Universal Robots PolyScope program: whisk_matcha.urp

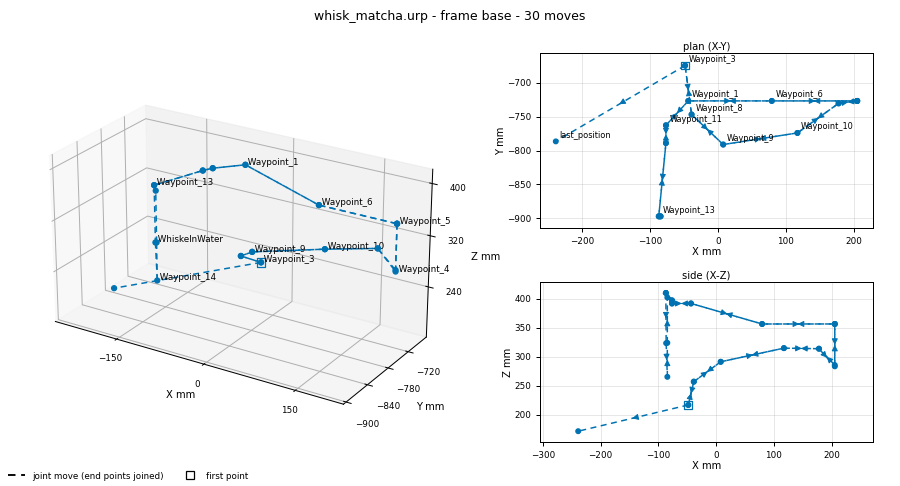
[picture p0: tool path of whisk_matcha.urp in frame base, 30 of 31 moves have a stored position in this frame; points joined in program order, loops and branches not executed]
Program whisk_matcha (installation=default directory=/programs/Matcha createdIn=5.12.6.1102099 lastSavedIn=5.12.6.1102099 robotSerialNumber=20215500597)
Calibrated DH parameters: a=[0.000193, -0.066673, -0.391568, -0.000012, 0.00005, 0]; d=[0.162643, -472.05677, 465.132521, 7.058239, 0.099746, 0.099582]; alpha=[1.571116, 0.00089, 0.003862, 1.569269, -1.569248, 0]; deltaTheta=[0, -1.413394, 7.628392, 0.068187, 0, -0.000001]
Robot Program (runOnlyOnce=true)
  URCap Gripper Activate (Robotiq_Grippers, Robotiq Inc.) dataModel(ResetAndActivateKey=false)
  URCap Gripper (Robotiq_Grippers, Robotiq Inc.) dataModel(position=14.117647058823529, force=0.0, speed=0.0, positionInDouble=14.117647058823529, forceInDouble=0.0, speedInDouble=0.0, slaveIds=[9], blocking=true)
  MoveJ speed 60 deg/s, acceleration 80 deg/s^2 (useActiveTCP=true) feature=Base
    Waypoint Waypoint (Variable): variable=matchaSpoonHome
    Waypoint Waypoint_3: TCP in base x=-48.218 y=-674.691 z=216.535 mm, rx=-1.0956 ry=1.5728 rz=-1.3161 rad; joints [49.709, -52.645, 74.816, -42.693, -23.853, -158.617] deg; TCP offset x=0 y=0 z=191.5 mm, rx=0 ry=0 rz=0 rad
    Waypoint Waypoint_8: TCP in base x=-38.666 y=-746.861 z=256.872 mm, rx=-0.5003 ry=1.6808 rz=-0.7695 rad; joints [54.631, -40.792, 48.492, -25.129, -23.202, -120.249] deg
    Waypoint Waypoint_9: TCP in base x=7.915 y=-791.123 z=291.294 mm, rx=0.1007 ry=1.6659 rz=-0.1248 rad; joints [60.017, -27.831, 19.708, -5.925, -22.495, -78.296] deg
    Waypoint Waypoint_10: TCP in base x=117.298 y=-774.028 z=314.897 mm, rx=0.8846 ry=1.446 rz=0.7971 rad; joints [67.52, -9.771, -20.402, 20.84, -21.505, -19.839] deg
    Waypoint Waypoint_2: TCP in base x=177.976 y=-730.441 z=313.913 mm, rx=1.2449 ry=1.2572 rz=1.2232 rad; joints [71.064, -1.234, -39.351, 33.486, -21.04, 7.782] deg
    Waypoint Waypoint_4: TCP in base x=205.418 y=-726.808 z=283.401 mm, rx=1.2448 ry=1.2573 rz=1.2232 rad; joints [73.018, 4.06, -46.322, 34.472, -19.107, 8.52] deg
  URCap Gripper (Robotiq_Grippers, Robotiq Inc.) dataModel(position=100.0, force=100.0, speed=64.0, positionInDouble=100.0, forceInDouble=100.0, speedInDouble=64.0, slaveIds=[9], blocking=true)
  MoveJ speed 60 deg/s, acceleration 80 deg/s^2 (useActiveTCP=true) feature=Base
    Waypoint Waypoint_5: TCP in base x=205.369 y=-726.831 z=356.753 mm, rx=1.2449 ry=1.2572 rz=1.2232 rad; joints [73.015, -6.018, -35.971, 34.181, -19.107, 8.543] deg
    Waypoint Waypoint_6: TCP in base x=79.554 y=-726.833 z=356.715 mm, rx=1.2449 ry=1.2572 rz=1.2232 rad; joints [63.962, -12.783, -20.178, 27.557, -28.074, 5.907] deg
    Waypoint Waypoint_1: TCP in base x=-43.538 y=-726.812 z=392.259 mm, rx=1.3602 ry=1.0584 rz=1.0356 rad; joints [53.28, -11.873, -28.744, 34.319, -24.003, 6.898] deg
    Waypoint Waypoint_11: TCP in base x=-76.429 y=-762.764 z=392.203 mm, rx=1.4056 ry=0.9656 rz=0.9484 rad; joints [51.982, -14.289, -22.965, 29.233, -18.545, 8.768] deg
    Waypoint Waypoint_18: TCP in base x=-76.468 y=-788.93 z=397.596 mm, rx=1.4283 ry=0.9152 rz=0.9007 rad; joints [52.819, -15.443, -21.159, 26.101, -14.083, 11.353] deg
    Waypoint Waypoint_13: TCP in base x=-87.04 y=-896.924 z=410.452 mm, rx=1.4774 ry=0.7933 rz=0.7855 rad; joints [56.392, -6.792, -35.013, -18.198, -2.939, 61.157] deg
  MoveJ speed 60 deg/s, acceleration 80 deg/s^2 (useActiveTCP=true) feature=Base
    Waypoint WhiskeInWater: TCP in base x=-86.518 y=-896.922 z=323.549 mm, rx=1.4625 ry=0.8327 rz=0.8228 rad; joints [56.475, -10.121, -18.162, -2.731, -4.889, 32.102] deg
    Waypoint Waypoint_14: TCP in base x=-84.466 y=-896.952 z=265.217 mm, rx=1.4624 ry=0.8326 rz=0.8227 rad; joints [56.595, -0.128, -30.65, -0.877, -4.787, 32.747] deg
    Wait Sleep waitTime=5
    Waypoint Waypoint_15: TCP in base x=-84.51 y=-896.917 z=324.084 mm, rx=1.4624 ry=0.8327 rz=0.8227 rad; joints [56.592, -9.392, -19.758, -2.594, -4.791, 32.83] deg
    Wait Sleep waitTime=5
  MoveJ speed 60 deg/s, acceleration 80 deg/s^2 (useActiveTCP=true) feature=Base
    Waypoint Waypoint_16: TCP in base x=-84.505 y=-896.935 z=402.694 mm, rx=1.4774 ry=0.7935 rz=0.7857 rad; joints [56.543, -4.6, -38.182, -19.515, -2.878, 63.454] deg
    Waypoint Waypoint_13: TCP in base x=-87.04 y=-896.924 z=410.452 mm, rx=1.4774 ry=0.7933 rz=0.7855 rad; joints [56.392, -6.792, -35.013, -18.198, -2.939, 61.157] deg
    Waypoint Waypoint_18: TCP in base x=-76.468 y=-788.93 z=397.596 mm, rx=1.4283 ry=0.9152 rz=0.9007 rad; joints [52.819, -15.443, -21.159, 26.101, -14.083, 11.353] deg
    Waypoint Waypoint_11: TCP in base x=-76.429 y=-762.764 z=392.203 mm, rx=1.4056 ry=0.9656 rz=0.9484 rad; joints [51.982, -14.289, -22.965, 29.233, -18.545, 8.768] deg
    Waypoint Waypoint_1: TCP in base x=-43.538 y=-726.812 z=392.259 mm, rx=1.3602 ry=1.0584 rz=1.0356 rad; joints [53.28, -11.873, -28.744, 34.319, -24.003, 6.898] deg
    Waypoint Waypoint_6: TCP in base x=79.554 y=-726.833 z=356.715 mm, rx=1.2449 ry=1.2572 rz=1.2232 rad; joints [63.962, -12.783, -20.178, 27.557, -28.074, 5.907] deg
    Waypoint Waypoint_5: TCP in base x=205.369 y=-726.831 z=356.753 mm, rx=1.2449 ry=1.2572 rz=1.2232 rad; joints [73.015, -6.018, -35.971, 34.181, -19.107, 8.543] deg
  MoveJ speed 60 deg/s, acceleration 80 deg/s^2 (useActiveTCP=true) feature=Base
    Waypoint Waypoint_5: TCP in base x=205.369 y=-726.831 z=356.753 mm, rx=1.2449 ry=1.2572 rz=1.2232 rad; joints [73.015, -6.018, -35.971, 34.181, -19.107, 8.543] deg
    Waypoint Waypoint_7: TCP in base x=205.328 y=-726.847 z=285.681 mm, rx=1.245 ry=1.2571 rz=1.2232 rad; joints [73.011, 3.773, -46.064, 34.504, -19.105, 8.521] deg
    URCap Gripper (Robotiq_Grippers, Robotiq Inc.) dataModel(position=52.549019607843135, force=100.0, speed=64.0, positionInDouble=52.549019607843135, forceInDouble=100.0, speedInDouble=64.0, slaveIds=[9], blocking=true)
    URCap Gripper (Robotiq_Grippers, Robotiq Inc.) dataModel(position=58.8235294117647, force=100.0, speed=64.0, positionInDouble=58.8235294117647, forceInDouble=100.0, speedInDouble=64.0, slaveIds=[9], blocking=true)
    URCap Gripper (Robotiq_Grippers, Robotiq Inc.) dataModel(position=14.117647058823529, force=0.0, speed=0.0, positionInDouble=14.117647058823529, forceInDouble=0.0, speedInDouble=0.0, slaveIds=[9], blocking=true)
  MoveJ speed 60 deg/s, acceleration 80 deg/s^2 (useActiveTCP=true) feature=Base
    Waypoint Waypoint_2: TCP in base x=177.976 y=-730.441 z=313.913 mm, rx=1.2449 ry=1.2572 rz=1.2232 rad; joints [71.064, -1.234, -39.351, 33.486, -21.04, 7.782] deg
    Waypoint Waypoint_10: TCP in base x=117.298 y=-774.028 z=314.897 mm, rx=0.8846 ry=1.446 rz=0.7971 rad; joints [67.52, -9.771, -20.402, 20.84, -21.505, -19.839] deg
    Waypoint Waypoint_9: TCP in base x=7.915 y=-791.123 z=291.294 mm, rx=0.1007 ry=1.6659 rz=-0.1248 rad; joints [60.017, -27.831, 19.708, -5.925, -22.495, -78.296] deg
    Waypoint Waypoint_8: TCP in base x=-38.666 y=-746.861 z=256.872 mm, rx=-0.5003 ry=1.6808 rz=-0.7695 rad; joints [54.631, -40.792, 48.492, -25.129, -23.202, -120.249] deg
    Waypoint Waypoint_3: TCP in base x=-48.218 y=-674.691 z=216.535 mm, rx=-1.0956 ry=1.5728 rz=-1.3161 rad; joints [49.709, -52.645, 74.816, -42.693, -23.853, -158.617] deg
    Waypoint last_position: TCP in base x=-238.783 y=-786.481 z=171.128 mm, rx=0.0287 ry=-2.2144 rz=2.2271 rad; joints [49.903, -56.994, 96.507, -40.117, 49.291, 179.673] deg
